SUBAPPLICATION Gesamtzaehler (* Subapplication Type *)
  (* Standard: 61499-2 *)
  (* Version 1.0, 2023-02-17, Franz *)
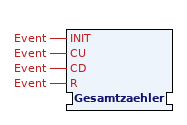
  EVENT_INPUT
    INIT; (* Initialization Request *)
    CU; (* Count Up *)
    CD; (* Count Down *)
    R; (* Reset *)
  END_EVENT
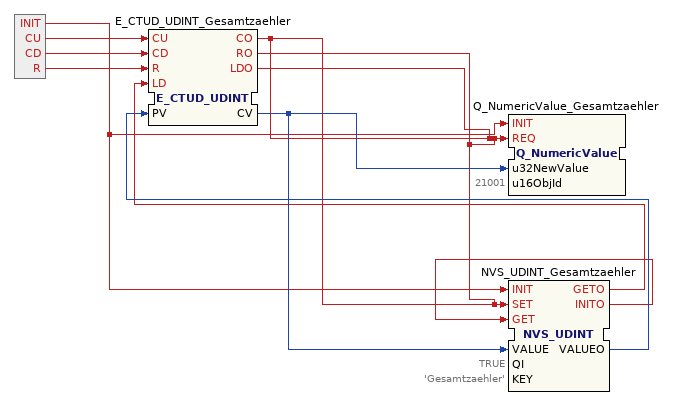
  FBS
    E_CTUD_UDINT_Gesamtzaehler : E_CTUD_UDINT;
    Q_NumericValue_Gesamtzaehler : Q_NumericValue(u16ObjId := 21001);
    NVS_UDINT_Gesamtzaehler : NVS_UDINT(QI := TRUE, KEY := 'Gesamtzaehler');
  END_FBS
  EVENT_CONNECTIONS
    INIT TO Q_NumericValue_Gesamtzaehler.INIT;
    E_CTUD_UDINT_Gesamtzaehler.CO TO Q_NumericValue_Gesamtzaehler.REQ;
    E_CTUD_UDINT_Gesamtzaehler.RO TO Q_NumericValue_Gesamtzaehler.REQ;
    E_CTUD_UDINT_Gesamtzaehler.LDO TO Q_NumericValue_Gesamtzaehler.REQ;
    CU TO E_CTUD_UDINT_Gesamtzaehler.CU;
    CD TO E_CTUD_UDINT_Gesamtzaehler.CD;
    R TO E_CTUD_UDINT_Gesamtzaehler.R;
    INIT TO NVS_UDINT_Gesamtzaehler.INIT;
    E_CTUD_UDINT_Gesamtzaehler.CO TO NVS_UDINT_Gesamtzaehler.SET;
    E_CTUD_UDINT_Gesamtzaehler.RO TO NVS_UDINT_Gesamtzaehler.SET;
    NVS_UDINT_Gesamtzaehler.GETO TO E_CTUD_UDINT_Gesamtzaehler.LD;
    NVS_UDINT_Gesamtzaehler.INITO TO NVS_UDINT_Gesamtzaehler.GET;
  END_CONNECTIONS
  DATA_CONNECTIONS
    E_CTUD_UDINT_Gesamtzaehler.CV TO Q_NumericValue_Gesamtzaehler.u32NewValue;
    E_CTUD_UDINT_Gesamtzaehler.CV TO NVS_UDINT_Gesamtzaehler.VALUE;
    NVS_UDINT_Gesamtzaehler.VALUEO TO E_CTUD_UDINT_Gesamtzaehler.PV;
  END_CONNECTIONS
END_SUBAPPLICATION
